// TIA Portal V16 export
// export: Created 2019-09-22T11:06:10.8135808Z, ExportSetting WithDefaults, DisplayName Totally Integrated Automation Portal, DisplayVersion V16, DisplayName TIA Portal Version Control Interface, DisplayVersion V16, DisplayName TIA Portal Openness, DisplayVersion V16, DisplayName STEP 7 Professional, DisplayVersion V16, DisplayName SIMATIC Energy Suite, DisplayVersion V16, DisplayName STEP 7 Safety, DisplayVersion V16, DisplayName WinCC Professional, DisplayVersion V16, DisplayName SIMATIC Visualization Architect, DisplayVersion V16
TYPE "typeShowIoSystem"
// stored: IsFailsafeCompliant false
   STRUCT
      device { S7_SetPoint := 'True'} : Array[1.."MAX_DEVICES_SYSTEM"] of "typeShowDevice";   // devices informations
   END_STRUCT;
END_TYPE
